VAR_GLOBAL CONSTANT
	MAX_D_OUT	: INT := 100;
END_VAR

(* stored: Version 1.1.0.1, ProductVersion 3.1.0.36
   GVL IO_DigiOut_Parameters: Id {722d774b-12ba-4072-887c-d802afd66bd2}, ParameterList True *)
